PROGRAM StartStopSequence_CC1Test
VAR_INPUT
	start : BOOL := FALSE;
	setSpeedDuration : TIME := T#0S;
	autoAdvance : BOOL := TRUE;
END_VAR
VAR_OUTPUT
	startTimes : ARRAY[1..50] OF ULINT;
	endTimes : ARRAY[1..50] OF ULINT;

	P9999Atubing : ARRAY[1..50] OF INT;
	P9999Btubing : ARRAY[1..50] OF INT;
END_VAR
VAR
	i : UINT := 0; // index
	n : UINT := 25;
	t : LREAL := 0.0;
	tol : LREAL := 5.0;
	spTotal : ARRAY [1..50] OF LREAL := [100.0,100.0,100.0,0.0,0.0,0.0,0.0,0.0,0.0,0.0,0.0,0.0,0.0,0.0,0.0,0.0,0.0,0.0,0.0,0.0,0.0,0.0,0.0,0.0, 0.0,
									0.0,0.0,0.0,0.0,0.0,0.0,0.0,0.0,0.0,0.0,0.0,0.0,0.0,0.0,0.0,0.0,0.0,0.0,0.0,0.0,0.0,0.0,0.0,0.0,0.0];
	//spTotal : ARRAY [1..50] OF LREAL := [100.0, 150.0, 200.0, 300.0, 150.0, 100.0, 80.0, 80.0, 90.0, 100.0, 
    //                                110.0, 120.0, 130.0, 140.0, 150.0, 0.0, 0.0, 0.0,
    //                                0.0, 0.0, 0.0, 0.0, 0.0, 0.0,
	//								0.0,0.0,0.0,0.0,0.0,0.0,0.0,0.0,0.0,0.0,0.0,0.0,0.0,0.0,0.0,0.0,0.0,0.0,0.0,0.0,0.0,0.0,0.0,0.0];
	spConc : ARRAY [1..50] OF LREAL := [1.0, 1.0, 1.0, 1.0, 1.0, 1.0, 1.0, 1.0, 1.0, 1.0, 
                                    1.0, 1.0, 1.0, 1.0, 1.0, 0.0, 0.0, 0.0,
                                    0.0, 0.0, 0.0, 0.0, 0.0, 0.0,
									0.0,0.0,0.0,0.0,0.0,0.0,0.0,0.0,0.0,0.0,0.0,0.0,0.0,0.0,0.0,0.0,0.0,0.0,0.0,0.0,0.0,0.0,0.0,0.0];
	stopTime : ARRAY [1..50] OF TIME := [T#0.5M, T#0.5M, T#0.5M, T#10.0M, T#15.0M, T#30.0M, T#60.0M, T#120.0M, T#1.0M, T#1.0M, 
                                    T#1.0M, T#1.0M, T#1.0M, T#1.0M, T#1.0M, T#0.0M, T#0.0M, T#0.0M,
                                    T#0.0M, T#0.0M, T#0.0M, T#0.0M, T#0.0M, T#0.0M,
									T#0.0M,T#0.0M,T#0.0M,T#0.0M,T#0.0M,T#0.0M,T#0.0M,T#0.0M,T#0.0M,T#0.0M,T#0.0M,T#0.0M,T#0.0M,
									T#0.0M,T#0.0M,T#0.0M,T#0.0M,T#0.0M,T#0.0M,T#0.0M,T#0.0M,T#0.0M,T#0.0M,T#0.0M];
	runTime : ARRAY [1..50] OF TIME := [T#0.1M, T#0.1M, T#0.1M, T#1.0M, T#1.0M, T#1.0M, T#1.0M, T#1.0M, T#1.0M, T#1.0M, 
                                    T#1.0M, T#1.0M, T#1.0M, T#1.0M, T#1.0M, T#0.0M, T#0.0M, T#0.0M,
                                    T#0.0M, T#0.0M, T#0.0M, T#0.0M, T#0.0M, T#0.0M,
									T#0.0M,T#0.0M,T#0.0M,T#0.0M,T#0.0M,T#0.0M,T#0.0M,T#0.0M,T#0.0M,T#0.0M,T#0.0M,T#0.0M,T#0.0M,
									T#0.0M,T#0.0M,T#0.0M,T#0.0M,T#0.0M,T#0.0M,T#0.0M,T#0.0M,T#0.0M,T#0.0M,T#0.0M];
	
	setSpeed : SFCStepType;
	runTest : SFCStepType;
	recordTest : SFCStepType;
END_VAR

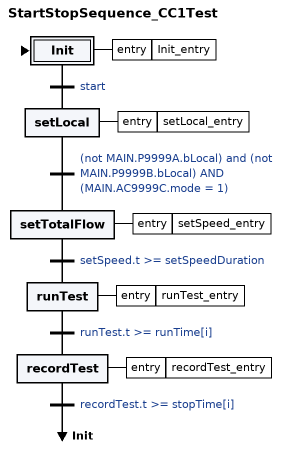
INITIAL_STEP Init:
    Init_entry(P1);  // entry action
END_STEP
TRANSITION FROM Init TO setLocal
    := start;
END_TRANSITION
STEP setLocal:
    setLocal_entry(P1);  // entry action
END_STEP
TRANSITION FROM setLocal TO setTotalFlow
    := (not MAIN.P9999A.bLocal) and (not MAIN.P9999B.bLocal) AND (MAIN.AC9999C.mode = 1);
END_TRANSITION
STEP setTotalFlow:
    setSpeed_entry(P1);  // entry action
END_STEP
TRANSITION FROM setTotalFlow TO runTest
    := setSpeed.t >= setSpeedDuration;
END_TRANSITION
STEP runTest:
    runTest_entry(P1);  // entry action
END_STEP
TRANSITION FROM runTest TO recordTest
    := runTest.t >= runTime[i];
END_TRANSITION
STEP recordTest:
    recordTest_entry(P1);  // entry action
END_STEP
TRANSITION FROM recordTest TO Init
    := recordTest.t >= stopTime[i];
END_TRANSITION

ACTION recordTest_entry:
endTimes[i] := unixTime;
MAIN.AC9999C.c.rq := 0; // set flow to 0 to stop pumps
t := DWORD_TO_LREAL(TIME_TO_DWORD(runTime[i]))/1000.0/60.0;

IF NOT autoAdvance THEN
	start := FALSE;
END_IF
END_ACTION

ACTION runTest_entry:
MAIN.MTSendString := 'SIR$0D$0A';
startTimes[i] := unixTime;
END_ACTION

ACTION resetTotals_entry:
MAIN.fbFQ9999A.resetRQ := TRUE;
MAIN.fbFQ9999B.resetRQ := TRUE;
MAIN.fbFQ9999C.resetRQ := TRUE;
MAIN.MTSendString := 'ZI$0D$0A';
MAIN.logActive := TRUE;
END_ACTION

ACTION setLocal_entry:
IF MAIN.P9999A.bLocal THEN
	MAIN.P9999A.nLocal_RQ := 0;  //put pump in remote
END_IF
IF MAIN.P9999B.bLocal THEN
	MAIN.P9999B.nLocal_RQ := 0;  //put pump in remote
END_IF

IF MAIN.AC9999C.mode <> 1 THEN 
	MAIN.AC9999C.mode := 1; // concentration control in auto
	MAIN.AC9999C.c.rq := 0; // set initial total flow
	MAIN.AC9999C.conc.rq := 1.0; // set initial concentration
	
END_IF
END_ACTION

ACTION setSpeed_entry:
i := i + 1;
startTimes[i] := 0;
endTimes[i] := 0;

MAIN.AC9999C.c.rq := spTotal[i];
MAIN.AC9999C.conc.rq := spConc[i];

P9999Atubing[i] := MAIN.P9999A.nTubeSize;
P9999Btubing[i] := MAIN.P9999B.nTubeSize;
END_ACTION

ACTION Init_entry:
IF i >= n THEN
	MAIN.AC9999C.mode := 0; // concentration control in manual
	MAIN.P9999A.nRun_RQ := 0; //stop pump
	MAIN.P9999B.nRun_RQ := 0; //stop pump
	start := FALSE;
	i := 0;
END_IF
MAIN.logActive := FALSE;
END_ACTION

END_PROGRAM

(* stored: Version 1.1.0.1, ProductVersion 3.1.0.36
   POU StartStopSequence_CC1Test: Id {14f49013-d3dd-4205-a8dc-c80c72f3680d}, SpecialFunc None
   Action recordTest_entry: Id {40fc5ea3-b802-42d8-8a80-7ede4ca07f16}
   Action runTest_entry: Id {4bb8c9c0-c090-4232-b342-273cde756878}
   Action resetTotals_entry: Id {556a9648-f35c-48e8-9a41-92303e3ecb5b}
   Action setLocal_entry: Id {80608a6b-c3dd-4fea-962b-2854f789f25d}
   Action setSpeed_entry: Id {8a12c593-cb81-4fa6-ba63-be9bfd1c77c2}
   Action Init_entry: Id {ecf34ce4-3fcf-409c-8fbb-d0faa82d51d8} *)
